// TwinCAT 3 PLC project lclc_plc_neh_n2
// ProgramVersion: 3.1.4022.7
// libraries:
//   LCLS General, * (SLAC)
//   Tc2_Standard, * (Beckhoff Automation GmbH)
//   Tc2_System, * (Beckhoff Automation GmbH)
//   Tc3_Module, * (Beckhoff Automation GmbH)
// project tree:
//   DUTs/ E_MAIN_STATE_MACHINE.TcDUT, E_LED_MODES.TcDUT, E_VALVE_RELAY_STATES.TcDUT
//   / PlcTask.TcTTO
//   POUs/ FB_LED_TOWER.TcPOU, FB_N2.TcPOU, FB_VALVE_RELAY.TcPOU, MAIN.TcPOU
// real-time tasks:
//   TASK PlcTask: cycle T#10ms, priority 20, ADS port 350
// I/O:
//   DEVICE Device 1 (EtherCAT), AmsNetId 192.168.0.100.2.1
//     Term 1 (EK1200) [EK1200-5000 EtherCAT Power supply (2A E-Bus)]
//       Term 2 (EL3052) [EL3052 2Ch. Ana. Input 4-20mA]
//       Term 3 (EL3052) [EL3052 2Ch. Ana. Input 4-20mA]
//       Term 4 (EL3054) [EL3054 4Ch. Ana. Input 4-20mA]
//       Term 5 (EL2624) [EL2624 4Ch. Relay Output, NO (125V AC / 30V DC)]
//       Term 6 (EL1004)
//       Term 14 (EL1004)
//       Term 7 (EL9011)
// variable links:
//   lclc_plc_neh_n2 Instance <-> Device 1 (EtherCAT)/Term 1 (EK1200)/Term 14 (EL1004)
//     PlcTask Inputs/MAIN.fbN2_Left.fbValveRelay.bCloseRBV <-> Channel 1/Input
//     PlcTask Inputs/MAIN.fbN2_Left.fbValveRelay.bMovingRBV <-> Channel 3/Input
//     PlcTask Inputs/MAIN.fbN2_Left.fbValveRelay.bOpenRBV <-> Channel 2/Input
//   lclc_plc_neh_n2 Instance <-> Device 1 (EtherCAT)/Term 1 (EK1200)/Term 2 (EL3052)
//     PlcTask Inputs/MAIN.fbN2_Left.rawInputmA <-> AI Standard Channel 1/Value
//     PlcTask Inputs/MAIN.fbN2_Right.rawInputmA <-> AI Standard Channel 2/Value
//   lclc_plc_neh_n2 Instance <-> Device 1 (EtherCAT)/Term 1 (EK1200)/Term 3 (EL3052)
//     PlcTask Inputs/MAIN.fbN2_Left.iPressRaw <-> AI Standard Channel 1/Value
//     PlcTask Inputs/MAIN.fbN2_Right.iPressRaw <-> AI Standard Channel 2/Value
//   lclc_plc_neh_n2 Instance <-> Device 1 (EtherCAT)/Term 1 (EK1200)/Term 5 (EL2624)
//     PlcTask Outputs/MAIN.fbN2_Left.fbValveRelay.rawOutputRelayChan1 <-> Channel 3/Output
//     PlcTask Outputs/MAIN.fbN2_Left.fbValveRelay.rawOutputRelayChan3 <-> Channel 4/Output
//     PlcTask Outputs/MAIN.fbN2_Right.fbValveRelay.rawOutputRelayChan1 <-> Channel 1/Output
//     PlcTask Outputs/MAIN.fbN2_Right.fbValveRelay.rawOutputRelayChan3 <-> Channel 2/Output
//   lclc_plc_neh_n2 Instance <-> Device 1 (EtherCAT)/Term 1 (EK1200)/Term 6 (EL1004)
//     PlcTask Inputs/MAIN.fbN2_Right.fbValveRelay.bCloseRBV <-> Channel 1/Input
//     PlcTask Inputs/MAIN.fbN2_Right.fbValveRelay.bMovingRBV <-> Channel 3/Input
//     PlcTask Inputs/MAIN.fbN2_Right.fbValveRelay.bOpenRBV <-> Channel 2/Input

CONFIGURATION lclc_plc_neh_n2
    RESOURCE PLC ON TwinCAT3
        TASK PlcTask(INTERVAL := T#10ms, PRIORITY := 20);
        PROGRAM MAIN WITH PlcTask : MAIN;
    END_RESOURCE
END_CONFIGURATION

// ---- DUTs/E_MAIN_STATE_MACHINE.TcDUT
{attribute 'qualified_only'}
{attribute 'strict'}
TYPE E_MAIN_STATE_MACHINE :
(
    INIT := 0,
    NOMINAL := 1,
    EXCHANGE_MODE := 2,
    BUTTON_WAIT := 3

);
END_TYPE

// ---- DUTs/E_LED_MODES.TcDUT
{attribute 'qualified_only'}
{attribute 'strict'}
TYPE E_LED_MODES :
(
    OFF := 0,
    GREEN := 1,
    YELLOW := 2,
    RED := 3
);
END_TYPE

// ---- DUTs/E_VALVE_RELAY_STATES.TcDUT
{attribute 'qualified_only'}
{attribute 'strict'}
TYPE E_VALVE_RELAY_STATES :
(
    INIT := 0,
    NOMINAL := 1,
    ACTUATE := 2,
    WAIT := 3
);
END_TYPE

// ---- POUs/MAIN.TcPOU
PROGRAM MAIN
VAR
    {attribute 'pytmc' := 'pv: KFE:N2:01'}
    {attribute 'TcLinkTo' := '
        .rawInputmA := TIID^Device 1 (EtherCAT)^Term 1 (EK1200)^Term 2 (EL3052)^AI Standard Channel 1^Value;
        .iPressRaw := TIID^Device 1 (EtherCAT)^Term 1 (EK1200)^Term 3 (EL3052)^AI Standard Channel 1^Value;
        .fbValveRelay.rawOutputRelayChan1 := TIID^Device 1 (EtherCAT)^Term 1 (EK1200)^Term 5 (EL2624)^Channel 3^Output;
        .fbValveRelay.rawOutputRelayChan3 := TIID^Device 1 (EtherCAT)^Term 1 (EK1200)^Term 5 (EL2624)^Channel 4^Output;
        .fbValveRelay.bCloseRBV := TIID^Device 1 (EtherCAT)^Term 1 (EK1200)^Term 14 (EL1004)^Channel 1^Input;
        .fbValveRelay.bOpenRBV := TIID^Device 1 (EtherCAT)^Term 1 (EK1200)^Term 14 (EL1004)^Channel 2^Input;
        .fbValveRelay.bMovingRBV := TIID^Device 1 (EtherCAT)^Term 1 (EK1200)^Term 14 (EL1004)^Channel 3^Input;

    '}
    fbN2_Left : FB_N2;

        {attribute 'pytmc' := 'pv: KFE:N2:02'}
    {attribute 'TcLinkTo' := '
        .rawInputmA := TIID^Device 1 (EtherCAT)^Term 1 (EK1200)^Term 2 (EL3052)^AI Standard Channel 2^Value;
        .iPressRaw := TIID^Device 1 (EtherCAT)^Term 1 (EK1200)^Term 3 (EL3052)^AI Standard Channel 2^Value;
        .fbValveRelay.rawOutputRelayChan1 := TIID^Device 1 (EtherCAT)^Term 1 (EK1200)^Term 5 (EL2624)^Channel 1^Output;
        .fbValveRelay.rawOutputRelayChan3 := TIID^Device 1 (EtherCAT)^Term 1 (EK1200)^Term 5 (EL2624)^Channel 2^Output;
        .fbValveRelay.bCloseRBV := TIID^Device 1 (EtherCAT)^Term 1 (EK1200)^Term 6 (EL1004)^Channel 1^Input;
        .fbValveRelay.bOpenRBV := TIID^Device 1 (EtherCAT)^Term 1 (EK1200)^Term 6 (EL1004)^Channel 2^Input;
        .fbValveRelay.bMovingRBV := TIID^Device 1 (EtherCAT)^Term 1 (EK1200)^Term 6 (EL1004)^Channel 3^Input;

    '}
    fbN2_Right : FB_N2;

END_VAR

fbN2_Left(tActuateTime:=T#24h);
fbN2_Right(tActuateTime:= T#23h);

END_PROGRAM

// ---- POUs/FB_N2.TcPOU
FUNCTION_BLOCK FB_N2
VAR_INPUT
    tActuateTime : TIME;
END_VAR
VAR_OUTPUT
END_VAR
VAR

    rawInputmA AT %I*: INT;

    // WILL KEEP AS PVS FOR NOW, CAN BE PHYSICAL BUTTONS AT SOME POINT
    {attribute 'pytmc' := 'pv: START_EXCHANGE'}
    bInduceButton AT %I*	: BOOL;
    {attribute 'pytmc' := 'pv: FINISH_EXCHANGE'}
    bFinishExchangeButton AT %I*	: BOOL;

    {attribute 'pytmc' := 'pv: VALVE'}
    fbValveRelay 	: FB_VALVE_RELAY;
    fbLEDTower		: FB_LED_TOWER;

    {attribute 'pytmc' := '
        pv: MAX_MASS
        field: EGU lbs
    '}
    maxMass: LREAL;
    {attribute 'pytmc' := '
        pv: MIN_MASS
        field: EGU lbs
    '}
    minMass: LREAL;
    {attribute 'pytmc' := '
        pv: MASS
        field: EGU lbs
    '}
    fMassofGas: LREAL;
    fmA: LREAL;

    {attribute 'pytmc' := '
        pv: PRESSURE
        field: EGU psi/g
    '}
    fPress : LREAL;
    fPressMa : LREAL;
    iPressRaw AT %I*	: INT;

    // WILL NEED SOME SENSABLE DEFAULT HERE?
    {attribute 'pytmc' := '
        pv: MIN_PRESS_THRESHOLD
        field: EGU psi/g
    '}
    fMinPressureThresh 		: LREAL ;
    {attribute 'pytmc' := '
        pv: MIN_MASS_THRESHOLD
        field: EGU lbs
    '}
    fMinMassThresh			: LREAL;
    {attribute 'pytmc' := '
        pv: MASS_WARNING_THRESHOLD
        field: EGU lbs
    '}
    fWarningThresh: LREAL;
    //
    {attribute 'pytmc' := 'pv: LED'}
    eLEDMode : E_LED_MODES;
    bValveTimerQ : BOOL;
    bInit : BOOL := TRUE;

    {attribute 'pytmc' := '
        pv: STATE

    '}
    iState : E_MAIN_STATE_MACHINE  := E_MAIN_STATE_MACHINE.INIT;
    {attribute 'pytmc' := 'pv: LED_FLASH'}
    bFlashFlag : BOOL := FALSE;

END_VAR

IF bInit THEN
    maxMass := 1000;
    minMass := 0;
    bInit := FALSE;
END_IF

fbValveRelay(bTimerQ=>bValveTimerQ,tActuateTime:=tActuateTime);
fbLEDTower(eLEDMode := eLEDMode, tFlashInterval:= T#1s, bFlashing:=bFlashFlag);

fmA := (rawInputmA / 32768.0) * 16.0 + 4;
fMassofGas := (fmA - 4.0) / 16.0 * maxMass + minMass;

fPressMa := (iPressRaw / 32768.0) * 16.0 + 4;
fPress := (fPressMa - 4.0) / 16.0 * 500;

CASE iState OF
    E_MAIN_STATE_MACHINE.INIT: // INIT

    IF ((fPress > fMinPressureThresh) AND (fMassofGas > fMinMassThresh)) THEN
        fbValveRelay.ACTUATE_VALVE(TRUE);
    ELSE
        fbValveRelay.ACTUATE_VALVE(FALSE);
        eLEDMode := E_LED_MODES.YELLOW;
        bFlashFlag := TRUE;
    END_IF

    iState := E_MAIN_STATE_MACHINE.NOMINAL;
    eLEDMode := E_LED_MODES.GREEN;
    bFlashFlag := FALSE;

    E_MAIN_STATE_MACHINE.NOMINAL: // Nominal

    IF bInduceButton THEN
        eLEDMode := E_LED_MODES.YELLOW;
        bFlashFlag := TRUE;
        iState := E_MAIN_STATE_MACHINE.EXCHANGE_MODE;
        fbValveRelay.ACTUATE_VALVE(FALSE);
    END_IF

    IF  ((fPress < fMinPressureThresh) OR (fMassofGas < fMinMassThresh)) THEN
        // SOLID RED
        eLEDMode := E_LED_MODES.RED;
        bFlashFlag := FALSE;
        iState := E_MAIN_STATE_MACHINE.BUTTON_WAIT;
        fbValveRelay.ACTUATE_VALVE(FALSE);
    ELSE
        eLEDMode := E_LED_MODES.GREEN;
        bFlashFlag := FALSE;
    END_IF

    IF (fMassofGas < fWarningThresh) THEN
        // SOLID YELLOW
        eLEDMode := E_LED_MODES.YELLOW;
        bFlashFlag := FALSE;
    END_IF

    IF(bValveTimerQ) THEN
        eLEDMode := E_LED_MODES.RED;
        bFlashFlag := TRUE;
    END_IF

    E_MAIN_STATE_MACHINE.BUTTON_WAIT:
    IF bInduceButton THEN
        iState := E_MAIN_STATE_MACHINE.EXCHANGE_MODE;
        eLEDMode := E_LED_MODES.YELLOW;
        bFlashFlag := TRUE;
        fbValveRelay.ACTUATE_VALVE(FALSE);
    END_IF

    E_MAIN_STATE_MACHINE.EXCHANGE_MODE: // EXCHANGE MODE
    IF (bInduceButton) THEN
        // FLASHING RED
        eLEDMode := E_LED_MODES.RED;
        bFlashFlag := TRUE;
    END_IF
    IF  ((bFinishExchangeButton)) THEN
        iState := E_MAIN_STATE_MACHINE.INIT;
        // SOLID GREEN
        eLEDMode := E_LED_MODES.GREEN;
        bFlashFlag := FALSE;

        // RESET BUTTON PRESSES
        bInduceButton := FALSE;
        bFinishExchangeButton := FALSE;
    END_IF

END_CASE

END_FUNCTION_BLOCK

// ---- POUs/FB_VALVE_RELAY.TcPOU
FUNCTION_BLOCK FB_VALVE_RELAY
VAR_IN_OUT
    tActuateTime : TIME ;
END_VAR
VAR_INPUT
END_VAR
VAR_OUTPUT
    bTimerQ : BOOL;
END_VAR
VAR
    {attribute 'pytmc' := 'pv: OPN_SW'}
    b_open : BOOL; // control variable
    // EL2624 Relayu Logic Here

    rawOutputRelayChan1 AT %Q*: BOOL;
    rawOutputRelayChan3 AT %Q*: BOOL;
    bCloseRBV AT %I* : BOOL;
    bOpenRBV AT %I* : BOOL;
    bMovingRBV AT %I* : BOOL;
    iState: E_VALVE_RELAY_STATES := E_VALVE_RELAY_STATES.INIT;
    fbValveTimer : TON;
END_VAR


fbValveTimer(IN:=TRUE, PT:=tActuateTime);

CASE iState OF
    E_VALVE_RELAY_STATES.INIT: // INIT
    IF fbValveTimer.Q THEN ACTUATE_VALVE(TRUE); END_IF
    fbValveTimer(IN:=FALSE); //RESTART TIMER
    iState := E_VALVE_RELAY_STATES.NOMINAL;

    E_VALVE_RELAY_STATES.NOMINAL: // NOMINAL
    ACTUATE_VALVE(b_open);

    // ONLY ACTUATE VALVE IF ITS OPEN
    IF fbValveTimer.Q AND bOpenRBV AND NOT bCloseRBV THEN
        iState := E_VALVE_RELAY_STATES.ACTUATE;
    ELSIF fbValveTimer.Q AND NOT bOpenRBV AND bCloseRBV THEN
        fbValveTimer(IN:=FALSE); //RESTART TIMER
    END_IF


    E_VALVE_RELAY_STATES.ACTUATE: // Do the opposite of current valve state
    ACTUATE_VALVE(FALSE);
    IF bMovingRBV THEN iState := E_VALVE_RELAY_STATES.WAIT; END_IF; // Only transition when we have started to move

    E_VALVE_RELAY_STATES.WAIT: // Go back to init to reset timer and return valve to previous state.
    IF NOT bMovingRBV THEN iState := E_VALVE_RELAY_STATES.INIT; END_IF;

END_CASE

bTimerQ := fbValveTimer.Q;

METHOD ACTUATE_VALVE : BOOL
VAR_INPUT
    open: BOOL;
END_VAR
b_open := open;

IF b_open THEN
    rawOutputRelayChan1 := FALSE;
    rawOutputRelayChan3 := TRUE;
ELSE
    rawOutputRelayChan1 := TRUE;
    rawOutputRelayChan3 := FALSE;
END_IF

IF bMovingRBV THEN iState := E_VALVE_RELAY_STATES.WAIT; END_IF; // Only transition when we have started to move
END_METHOD

END_FUNCTION_BLOCK

// ---- POUs/FB_LED_TOWER.TcPOU
FUNCTION_BLOCK FB_LED_TOWER
VAR_INPUT
    eLEDMode : E_LED_MODES;
    tFlashInterval : TIME;
    bFlashing : BOOL := FALSE;

END_VAR
VAR_OUTPUT
END_VAR
VAR
    bGreenPin AT %I* : BOOL;
    bYellowPin AT %I* : BOOL;
    bRedPin AT %I* : BOOL;

    tLEDFLashTimerON : TON;
    tLEDFLashTimerOFF : TOF;


END_VAR

IF eLEDMode = E_LED_MODES.OFF THEN
    bGreenPin := FALSE;
    bYellowPin := FALSE;
    bRedPin := FALSE;
    RETURN;
END_IF

tLEDFLashTimerON(IN:=bFlashing, PT:=tFlashInterval);
tLEDFLashTimerOFF(IN:= NOT tLEDFLashTimerON.Q, PT:=tFlashInterval);

bGreenPin := FALSE;
bYellowPin := FALSE;
bRedPin := FALSE;

CASE eLEDMode OF
    E_LED_MODES.GREEN:
        bGreenPin := NOT bFlashing OR tLEDFLashTimerON.Q;
    E_LED_MODES.YELLOW:
        bYellowPin := NOT bFlashing OR tLEDFLashTimerON.Q;
        bRedPin := FALSE;
    E_LED_MODES.RED:
        bRedPin :=  NOT bFlashing OR tLEDFLashTimerON.Q;
END_CASE

IF NOT tLEDFLashTimerOFF.Q THEN
    tLEDFLashTimerON(IN:=FALSE);
END_IF

END_FUNCTION_BLOCK
